Fanuc KAREL source: kd00006.KL

-- PROVISIONAL review KL for V940-1; original PC SHA256 9769cb4164fce735e4a834b79c69105eea25169a61e229dd1c19ab7abce9fcab
-- Incomplete behavior may be omitted. Consult companion uncertainty JSON. Do not deploy.
PROGRAM KD00006
%NOLOCKGROUP
VAR
  I : INTEGER
  J : INTEGER
  B : BOOLEAN
  R : REAL
  S : STRING[80]
BEGIN
  -- V9_ZERO_TABLE_METADATA_HINT layout=0001; no indexed target words; source/name/runtime held
  -- UNRESOLVED_PC offsets 5-12; opcodes 9D,23
  -- UNRESOLVED_PC offsets 17-21; opcodes 7F
END KD00006
